// Mitsubishi GX Works2 project: 0709자동차후진   PLC: Q02/Q02H

PROGRAM MAIN
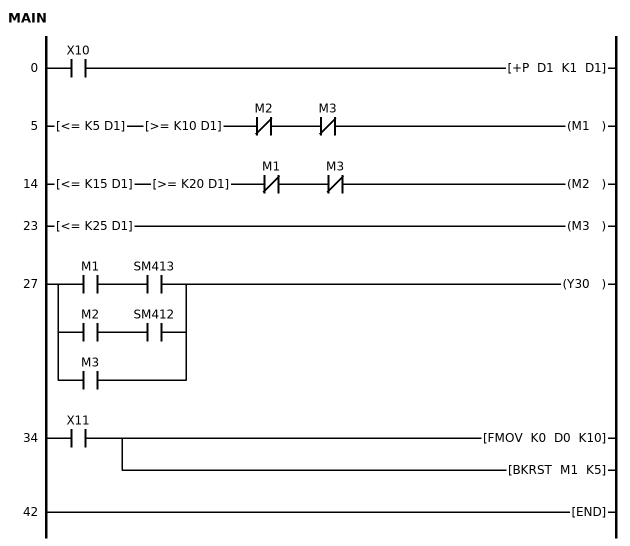
0     LD      X10
      +P      D1 K1 D1
5     LD<=    K5 D1
      AND>=   K10 D1
      ANI     M2
      ANI     M3
      OUT     M1
14    LD<=    K15 D1
      AND>=   K20 D1
      ANI     M1
      ANI     M3
      OUT     M2
23    LD<=    K25 D1
      OUT     M3
27    LD      M1
      AND     SM413
      LD      M2
      AND     SM412
      ORB
      OR      M3
      OUT     Y30
34    LD      X11
      FMOV    K0 D0 K10
      BKRST   M1 K5
42    END
END_PROGRAM
